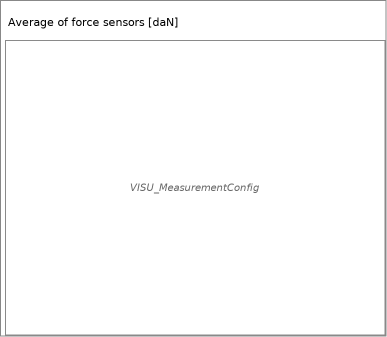
VISUALIZATION VISU_M1Config_Axial_AverageForce  // 387x337
VAR_IN_OUT
    editable : M1AxialSupportConfig;
	active : M1AxialSupportConfig;
END_VAR
    Frame (5,40 380x295)
        shows VISU_MeasurementConfig(active := active.mirrorAverageForce, editable := editable.mirrorAverageForce)
    Label (5,0 225x45), "Average of force sensors [daN]"
END_VISUALIZATION

(* stored: Version 1.1.0.1, ProductVersion 3.1.4019.2
   Visu VISU_M1Config_Axial_AverageForce: Id {2d0c6a99-032d-43c4-8f64-f86e3729ad36} *)
